// TIA Portal V19 export
TYPE "LEXCHANGETRAY_typeNgStrapManualCommands"
TITLE = exchangeTray_typeNgStrapManualCommands
// exchangeTray_typeNgStrapManualCommands related values
// stored: Access Published
   STRUCT
      resetCount { ExternalAccessible := 'False'; ExternalVisible := 'False'; ExternalWritable := 'False'} : Bool;   // Reset count manual command
      resetError { ExternalAccessible := 'False'; ExternalVisible := 'False'; ExternalWritable := 'False'} : Bool;   // Reset error manual command
      raiseError { ExternalAccessible := 'False'; ExternalVisible := 'False'; ExternalWritable := 'False'} : Bool;   // Raise error manual command
      simStart { ExternalAccessible := 'False'; ExternalVisible := 'False'; ExternalWritable := 'False'} : Bool;   // Start simulation manual command
      simOK { ExternalAccessible := 'False'; ExternalVisible := 'False'; ExternalWritable := 'False'} : Bool;   // Simulation OK manual command
   END_STRUCT;
END_TYPE
